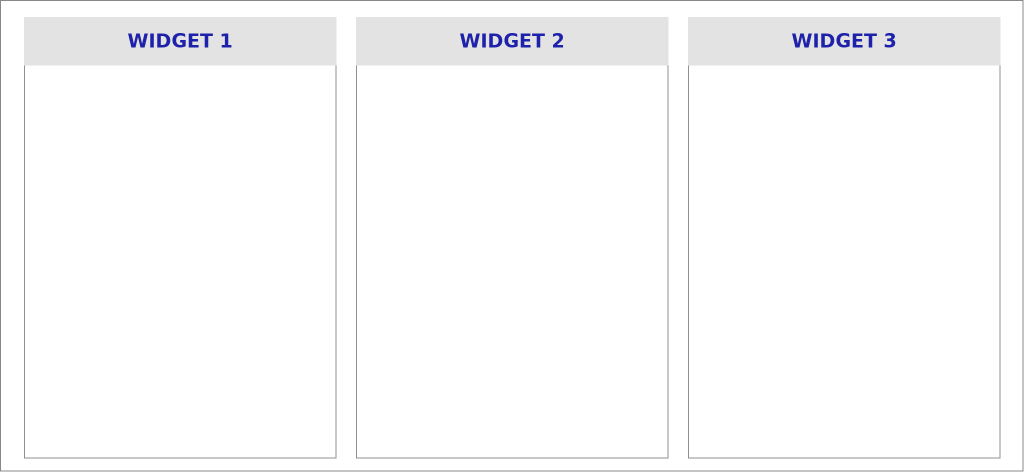
VISUALIZATION _000_Home  // 1024x472
    GroupBox (24,16 312x442)
        Rectangle (0,1 312x48), "WIDGET 1"
    GroupBox (356,16 312x442)
        Rectangle (0,1 312x48), "WIDGET 2"
    GroupBox (688,16 312x442)
        Rectangle (0,1 312x48), "WIDGET 3"
END_VISUALIZATION

(* stored: Version 1.1.0.1, ProductVersion 3.1.4022.18
   Visu _000_Home: Id {6bc88143-e34a-4cbb-879b-af85fb2d675f} *)
